ABB RAPID module: Rapid logo Inclinado.mod

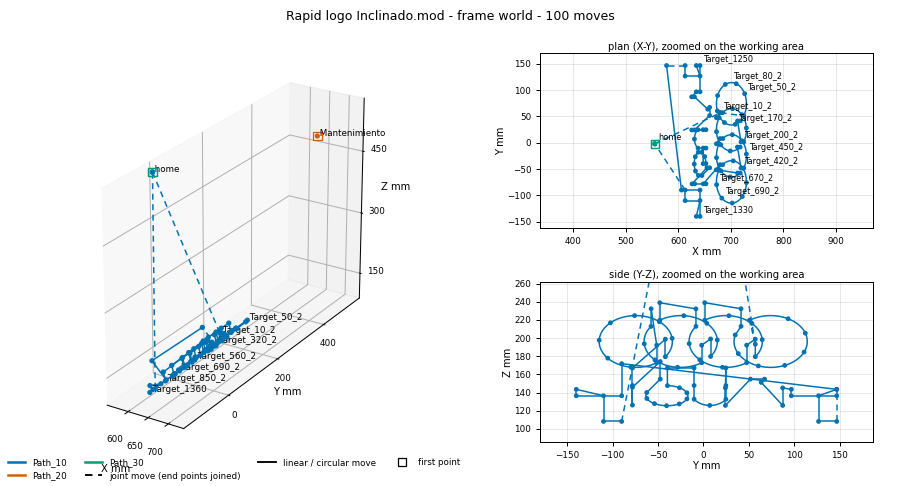
[picture p0: tool path of Rapid logo Inclinado.mod in frame world, 100 of 100 moves have a stored position in this frame; points joined in program order, loops and branches not executed]
MODULE Module1
    CONST robtarget Target_10_2:=[[-56.37355629,21.833194655,-12.40407904],[0.707106781,0,0,0.707106781],[0,0,-1,1],[9E+09,9E+09,9E+09,9E+09,9E+09,9E+09]];
    CONST robtarget Target_20_2:=[[-50.227,-27.838086869,0.000707115],[0.707106781,0,0,0.707106781],[0,0,-1,1],[9E+09,9E+09,9E+09,9E+09,9E+09,9E+09]];
    CONST robtarget Target_30_2:=[[-50.227,-27.838316171,0.001135326],[0.707106781,0,0,0.707106781],[0,0,-1,1],[9E+09,9E+09,9E+09,9E+09,9E+09,9E+09]];
    CONST robtarget Target_40_2:=[[-78.443,-34.755674334,0.002156228],[0.707106781,0,0,0.707106781],[0,0,-1,1],[9E+09,9E+09,9E+09,9E+09,9E+09,9E+09]];
    CONST robtarget Target_50_2:=[[-92.484,-30.22935476,0.001816803],[0.707106781,0,0,0.707106781],[0,0,-1,1],[9E+09,9E+09,9E+09,9E+09,9E+09,9E+09]];
    CONST robtarget Target_60_2:=[[-104.135,-20.748420193,0.00095273],[0.707106781,0,0,0.707106781],[0,0,-1,1],[9E+09,9E+09,9E+09,9E+09,9E+09,9E+09]];
    CONST robtarget Target_70_2:=[[-111.492,-7.712859409,0.000760167],[0.707106781,0,0,0.707106781],[0,0,-1,1],[9E+09,9E+09,9E+09,9E+09,9E+09,9E+09]];
    CONST robtarget Target_80_2:=[[-113.551,7.814084168,-0.000316037],[0.707106781,0,0,0.707106781],[0,0,-1,1],[9E+09,9E+09,9E+09,9E+09,9E+09,9E+09]];
    CONST robtarget Target_90_2:=[[-110.107,21.743448618,-0.000425835],[0.707106781,0,0,0.707106781],[0,0,-1,1],[9E+09,9E+09,9E+09,9E+09,9E+09,9E+09]];
    CONST robtarget Target_100_2:=[[-101.518,34.06976979,-0.001033142],[0.707106781,0,0,0.707106781],[0,0,-1,1],[9E+09,9E+09,9E+09,9E+09,9E+09,9E+09]];
    CONST robtarget Target_110_2:=[[-88.877,42.457578322,-0.001209673],[0.707106781,0,0,0.707106781],[0,0,-1,1],[9E+09,9E+09,9E+09,9E+09,9E+09,9E+09]];
    CONST robtarget Target_120_2:=[[-75.046,45.550294377,-0.000574222],[0.707106781,0,0,0.707106781],[0,0,-1,1],[9E+09,9E+09,9E+09,9E+09,9E+09,9E+09]];
    CONST robtarget Target_130_2:=[[-59.737,43.24160957,-0.001254548],[0.707106781,0,0,0.707106781],[0,0,-1,1],[9E+09,9E+09,9E+09,9E+09,9E+09,9E+09]];
    CONST robtarget Target_140_2:=[[-46.87,35.727016258,-0.000654802],[0.707106781,0,0,0.707106781],[0,0,-1,1],[9E+09,9E+09,9E+09,9E+09,9E+09,9E+09]];
    CONST robtarget Target_150_2:=[[-37.62,24.074953917,-0.00022001],[0.707106781,0,0,0.707106781],[0,0,-1,1],[9E+09,9E+09,9E+09,9E+09,9E+09,9E+09]];
    CONST robtarget Target_160_2:=[[-33.231,9.934106808,-0.000401667],[0.707106781,0,0,0.707106781],[0,0,-1,1],[9E+09,9E+09,9E+09,9E+09,9E+09,9E+09]];
    CONST robtarget Target_170_2:=[[-34.268,-4.941898461,0.000110514],[0.707106781,0,0,0.707106781],[0,0,-1,1],[9E+09,9E+09,9E+09,9E+09,9E+09,9E+09]];
    CONST robtarget Target_180_2:=[[-40.693,-18.501236857,0.089106304],[0.707106781,0,0,0.707106781],[0,0,-1,1],[9E+09,9E+09,9E+09,9E+09,9E+09,9E+09]];
    CONST robtarget Target_190_2:=[[-40.659,-28.454720515,-17.319460468],[0.707106781,0,0,0.707106781],[0,0,-1,1],[9E+09,9E+09,9E+09,9E+09,9E+09,9E+09]];
    CONST robtarget Target_200_2:=[[-0.697,-37.838908963,-17.319030487],[0.707106781,0,0,0.707106781],[0,0,-1,1],[9E+09,9E+09,9E+09,9E+09,9E+09,9E+09]];
    CONST robtarget Target_210_2:=[[-0.697,-27.838316171,0.001135326],[0.707106781,0,0,0.707106781],[0,0,-1,1],[9E+09,9E+09,9E+09,9E+09,9E+09,9E+09]];
    CONST robtarget Target_220_2:=[[-13.615,-33.787079032,0.001779373],[0.707106781,0,0,0.707106781],[0,0,-1,1],[9E+09,9E+09,9E+09,9E+09,9E+09,9E+09]];
    CONST robtarget Target_230_2:=[[-27.286,-34.931310202,0.001952004],[0.707106781,0,0,0.707106781],[0,0,-1,1],[9E+09,9E+09,9E+09,9E+09,9E+09,9E+09]];
    CONST robtarget Target_240_2:=[[-41.038,-31.199816129,0.000961671],[0.707106781,0,0,0.707106781],[0,0,-1,1],[9E+09,9E+09,9E+09,9E+09,9E+09,9E+09]];
    CONST robtarget Target_250_2:=[[-52.601,-22.954894729,0.001302226],[0.707106781,0,0,0.707106781],[0,0,-1,1],[9E+09,9E+09,9E+09,9E+09,9E+09,9E+09]];
    CONST robtarget Target_260_2:=[[-60.575,-11.244165105,0.000480163],[0.707106781,0,0,0.707106781],[0,0,-1,1],[9E+09,9E+09,9E+09,9E+09,9E+09,9E+09]];
    CONST robtarget Target_270_2:=[[-63.996,2.327231469,0.000364069],[0.707106781,0,0,0.707106781],[0,0,-1,1],[9E+09,9E+09,9E+09,9E+09,9E+09,9E+09]];
    CONST robtarget Target_280_2:=[[-62.487,16.549566353,-0.000316047],[0.707106781,0,0,0.707106781],[0,0,-1,1],[9E+09,9E+09,9E+09,9E+09,9E+09,9E+09]];
    CONST robtarget Target_290_2:=[[-56.39,28.971767635,-0.000857416],[0.707106781,0,0,0.707106781],[0,0,-1,1],[9E+09,9E+09,9E+09,9E+09,9E+09,9E+09]];
    CONST robtarget Target_300_2:=[[-56.367,19.00342355,-17.321167927],[0.707106781,0,0,0.707106781],[0,0,-1,1],[9E+09,9E+09,9E+09,9E+09,9E+09,9E+09]];
    CONST robtarget Target_310_2:=[[-46.834,28.340604975,-17.321014884],[0.707106781,0,0,0.707106781],[0,0,-1,1],[9E+09,9E+09,9E+09,9E+09,9E+09,9E+09]];
    CONST robtarget Target_320_2:=[[-46.834,38.341197767,-0.00084907],[0.707106781,0,0,0.707106781],[0,0,-1,1],[9E+09,9E+09,9E+09,9E+09,9E+09,9E+09]];
    CONST robtarget Target_330_2:=[[-33.859,44.305218974,-0.001065436],[0.707106781,0,0,0.707106781],[0,0,-1,1],[9E+09,9E+09,9E+09,9E+09,9E+09,9E+09]];
    CONST robtarget Target_340_2:=[[-20.239,45.433325791,-0.001165718],[0.707106781,0,0,0.707106781],[0,0,-1,1],[9E+09,9E+09,9E+09,9E+09,9E+09,9E+09]];
    CONST robtarget Target_350_2:=[[-6.223,41.574568908,-0.000596655],[0.707106781,0,0,0.707106781],[0,0,-1,1],[9E+09,9E+09,9E+09,9E+09,9E+09,9E+09]];
    CONST robtarget Target_360_2:=[[4.844,33.686749376,-0.000430885],[0.707106781,0,0,0.707106781],[-1,-1,0,1],[9E+09,9E+09,9E+09,9E+09,9E+09,9E+09]];
    CONST robtarget Target_370_2:=[[12.797,22.289578631,-0.000519591],[0.707106781,0,0,0.707106781],[-1,-1,0,1],[9E+09,9E+09,9E+09,9E+09,9E+09,9E+09]];
    CONST robtarget Target_380_2:=[[16.431,8.6200699,-0.000335384],[0.707106781,0,0,0.707106781],[-1,-1,0,1],[9E+09,9E+09,9E+09,9E+09,9E+09,9E+09]];
    CONST robtarget Target_390_2:=[[14.958,-6.043086672,0.000834231],[0.707106781,0,0,0.707106781],[-1,-1,0,1],[9E+09,9E+09,9E+09,9E+09,9E+09,9E+09]];
    CONST robtarget Target_400_2:=[[8.986,-18.294616208,0.000981918],[0.707106781,0,0,0.707106781],[-1,-1,0,1],[9E+09,9E+09,9E+09,9E+09,9E+09,9E+09]];
    CONST robtarget Target_410_2:=[[9.008,-28.264326332,-17.319694571],[0.707106781,0,0,0.707106781],[-1,-1,0,1],[9E+09,9E+09,9E+09,9E+09,9E+09,9E+09]];
    CONST robtarget Target_420_2:=[[48.833,-37.838908963,-17.319030487],[0.707106781,0,0,0.707106781],[-1,-1,0,1],[9E+09,9E+09,9E+09,9E+09,9E+09,9E+09]];
    CONST robtarget Target_430_2:=[[48.833,-27.838316171,0.001135326],[0.707106781,0,0,0.707106781],[-1,-1,0,1],[9E+09,9E+09,9E+09,9E+09,9E+09,9E+09]];
    CONST robtarget Target_440_2:=[[36.191,-33.714519443,0.001453804],[0.707106781,0,0,0.707106781],[-1,-1,0,1],[9E+09,9E+09,9E+09,9E+09,9E+09,9E+09]];
    CONST robtarget Target_450_2:=[[22.379,-34.942970463,0.00175625],[0.707106781,0,0,0.707106781],[-1,-1,0,1],[9E+09,9E+09,9E+09,9E+09,9E+09,9E+09]];
    CONST robtarget Target_460_2:=[[8.645,-31.272375718,0.001287239],[0.707106781,0,0,0.707106781],[-1,-1,0,1],[9E+09,9E+09,9E+09,9E+09,9E+09,9E+09]];
    CONST robtarget Target_470_2:=[[-2.93,-23.098281891,0.000953305],[0.707106781,0,0,0.707106781],[0,0,-1,1],[9E+09,9E+09,9E+09,9E+09,9E+09,9E+09]];
    CONST robtarget Target_480_2:=[[-10.814,-11.750850244,0.000893078],[0.707106781,0,0,0.707106781],[0,0,-1,1],[9E+09,9E+09,9E+09,9E+09,9E+09,9E+09]];
    CONST robtarget Target_490_2:=[[-14.498,2.811096116,0.000425657],[0.707106781,0,0,0.707106781],[0,0,-1,1],[9E+09,9E+09,9E+09,9E+09,9E+09,9E+09]];
    CONST robtarget Target_500_2:=[[-13.011,16.365002299,0.000015933],[0.707106781,0,0,0.707106781],[0,0,-1,1],[9E+09,9E+09,9E+09,9E+09,9E+09,9E+09]];
    CONST robtarget Target_510_2:=[[-7.137,28.586515175,-0.000121108],[0.707106781,0,0,0.707106781],[0,0,-1,1],[9E+09,9E+09,9E+09,9E+09,9E+09,9E+09]];
    CONST robtarget Target_520_2:=[[-7.137,18.585922383,-17.320286922],[0.707106781,0,0,0.707106781],[0,0,-1,1],[9E+09,9E+09,9E+09,9E+09,9E+09,9E+09]];
    CONST robtarget Target_530_2:=[[2.696,28.340604975,-17.321014884],[0.707106781,0,0,0.707106781],[0,0,-1,1],[9E+09,9E+09,9E+09,9E+09,9E+09,9E+09]];
    CONST robtarget Target_540_2:=[[2.696,38.341197767,-0.00084907],[0.707106781,0,0,0.707106781],[0,0,-1,1],[9E+09,9E+09,9E+09,9E+09,9E+09,9E+09]];
    CONST robtarget Target_550_2:=[[14.997,44.124253005,-0.000501529],[0.707106781,0,0,0.707106781],[-1,-1,0,1],[9E+09,9E+09,9E+09,9E+09,9E+09,9E+09]];
    CONST robtarget Target_560_2:=[[29.288,45.434191799,-0.001665747],[0.707106781,0,0,0.707106781],[-1,-1,0,1],[9E+09,9E+09,9E+09,9E+09,9E+09,9E+09]];
    CONST robtarget Target_570_2:=[[43.337,41.559310564,-0.001024336],[0.707106781,0,0,0.707106781],[-1,-1,0,1],[9E+09,9E+09,9E+09,9E+09,9E+09,9E+09]];
    CONST robtarget Target_580_2:=[[54.189,33.872679468,-0.000396886],[0.707106781,0,0,0.707106781],[-1,-1,0,1],[9E+09,9E+09,9E+09,9E+09,9E+09,9E+09]];
    CONST robtarget Target_590_2:=[[62.528,21.849622952,-0.000530122],[0.707106781,0,0,0.707106781],[-1,-1,0,1],[9E+09,9E+09,9E+09,9E+09,9E+09,9E+09]];
    CONST robtarget Target_600_2:=[[65.937,8.892951917,0.000300757],[0.707106781,0,0,0.707106781],[-1,-1,0,1],[9E+09,9E+09,9E+09,9E+09,9E+09,9E+09]];
    CONST robtarget Target_610_2:=[[64.517,-5.942742468,0.000632066],[0.707106781,0,0,0.707106781],[-1,-1,0,1],[9E+09,9E+09,9E+09,9E+09,9E+09,9E+09]];
    CONST robtarget Target_620_2:=[[58.496,-18.322400822,0.000858513],[0.707106781,0,0,0.707106781],[-1,-1,0,1],[9E+09,9E+09,9E+09,9E+09,9E+09,9E+09]];
    CONST robtarget Target_630_2:=[[58.383,-28.479773053,-17.318851916],[0.707106781,0,0,0.707106781],[-1,-1,0,1],[9E+09,9E+09,9E+09,9E+09,9E+09,9E+09]];
    CONST robtarget Target_640_2:=[[52.226,28.340604975,-17.321014884],[0.707106781,0,0,0.707106781],[-1,-1,0,1],[9E+09,9E+09,9E+09,9E+09,9E+09,9E+09]];
    CONST robtarget Target_650_2:=[[52.226,38.341197767,-0.00084907],[0.707106781,0,0,0.707106781],[-1,-1,0,1],[9E+09,9E+09,9E+09,9E+09,9E+09,9E+09]];
    CONST robtarget Target_660_2:=[[65.447,44.367484341,-0.001220779],[0.707106781,0,0,0.707106781],[-1,-1,0,1],[9E+09,9E+09,9E+09,9E+09,9E+09,9E+09]];
    CONST robtarget Target_670_2:=[[80.648,45.231271346,-0.001127368],[0.707106781,0,0,0.707106781],[-1,-1,0,1],[9E+09,9E+09,9E+09,9E+09,9E+09,9E+09]];
    CONST robtarget Target_680_2:=[[94.887,40.510959505,-0.000785768],[0.707106781,0,0,0.707106781],[-1,-1,0,1],[9E+09,9E+09,9E+09,9E+09,9E+09,9E+09]];
    CONST robtarget Target_690_2:=[[106.195,31.179608209,-0.000840934],[0.707106781,0,0,0.707106781],[-1,-1,0,1],[9E+09,9E+09,9E+09,9E+09,9E+09,9E+09]];
    CONST robtarget Target_700_2:=[[113.612,17.854675076,0.000153874],[0.707106781,0,0,0.707106781],[-1,-1,0,1],[9E+09,9E+09,9E+09,9E+09,9E+09,9E+09]];
    CONST robtarget Target_710_2:=[[115.581,3.23046335,0.000776639],[0.707106781,0,0,0.707106781],[-1,-1,0,1],[9E+09,9E+09,9E+09,9E+09,9E+09,9E+09]];
    CONST robtarget Target_720_2:=[[112.232,-10.957390781,0.001178007],[0.707106781,0,0,0.707106781],[-1,-1,0,1],[9E+09,9E+09,9E+09,9E+09,9E+09,9E+09]];
    CONST robtarget Target_730_2:=[[103.201,-23.874250963,0.000962006],[0.707106781,0,0,0.707106781],[-1,-1,0,1],[9E+09,9E+09,9E+09,9E+09,9E+09,9E+09]];
    CONST robtarget Target_740_2:=[[90.94,-31.928278149,0.001253355],[0.707106781,0,0,0.707106781],[-1,-1,0,1],[9E+09,9E+09,9E+09,9E+09,9E+09,9E+09]];
    CONST robtarget Target_750_2:=[[76.607,-35.064403142,0.001432857],[0.707106781,0,0,0.707106781],[-1,-1,0,1],[9E+09,9E+09,9E+09,9E+09,9E+09,9E+09]];
    CONST robtarget Target_760_2:=[[62.223,-32.908533711,0.001434457],[0.707106781,0,0,0.707106781],[-1,-1,0,1],[9E+09,9E+09,9E+09,9E+09,9E+09,9E+09]];
    CONST robtarget Target_770_2:=[[49.279,-25.574906369,0.001398618],[0.707106781,0,0,0.707106781],[-1,-1,0,1],[9E+09,9E+09,9E+09,9E+09,9E+09,9E+09]];
    CONST robtarget Target_780_2:=[[39.611,-13.556813975,0.000933947],[0.707106781,0,0,0.707106781],[-1,-1,0,1],[9E+09,9E+09,9E+09,9E+09,9E+09,9E+09]];
    CONST robtarget Target_790_2:=[[35.255,0.363122261,0.000494345],[0.707106781,0,0,0.707106781],[-1,-1,0,1],[9E+09,9E+09,9E+09,9E+09,9E+09,9E+09]];
    CONST robtarget Target_800_2:=[[36.202,15.191620477,-0.00030082],[0.707106781,0,0,0.707106781],[-1,-1,0,1],[9E+09,9E+09,9E+09,9E+09,9E+09,9E+09]];
    CONST robtarget Target_810_2:=[[42.65,28.945349059,-0.000614842],[0.707106781,0,0,0.707106781],[-1,-1,0,1],[9E+09,9E+09,9E+09,9E+09,9E+09,9E+09]];
    CONST robtarget Target_820_2:=[[42.65,18.944756267,-17.320780656],[0.707106781,0,0,0.707106781],[-1,-1,0,1],[9E+09,9E+09,9E+09,9E+09,9E+09,9E+09]];
    CONST robtarget Target_830_2:=[[78.968,63.836225874,-17.322010862],[0.707106781,0,0,0.707106781],[-1,-1,0,1],[9E+09,9E+09,9E+09,9E+09,9E+09,9E+09]];
    CONST robtarget Target_840_2:=[[78.968,73.836818666,-0.001845049],[0.707106781,0,0,0.707106781],[-1,-1,0,1],[9E+09,9E+09,9E+09,9E+09,9E+09,9E+09]];
    CONST robtarget Target_850_2:=[[78.968,104.377324543,-0.003182388],[0.707106781,0,0,0.707106781],[-1,-1,0,1],[9E+09,9E+09,9E+09,9E+09,9E+09,9E+09]];
    CONST robtarget Target_860_2:=[[78.968,93.82340557,-17.323718301],[0.707106781,0,0,0.707106781],[-1,-1,0,1],[9E+09,9E+09,9E+09,9E+09,9E+09,9E+09]];
    CONST robtarget Target_870_2:=[[48.351,53.873158678,-17.322208436],[0.707106781,0,0,0.707106781],[-1,-1,0,1],[9E+09,9E+09,9E+09,9E+09,9E+09,9E+09]];
    CONST robtarget Target_880_2:=[[48.351,63.87375147,-0.002042622],[0.707106781,0,0,0.707106781],[-1,-1,0,1],[9E+09,9E+09,9E+09,9E+09,9E+09,9E+09]];
    CONST robtarget Target_890_2:=[[63.169,84.713777945,-0.002771169],[0.707106781,0,0,0.707106781],[-1,-1,0,1],[9E+09,9E+09,9E+09,9E+09,9E+09,9E+09]];
    CONST robtarget Target_900_2:=[[64.162,89.365128281,-0.002555273],[0.707106781,0,0,0.707106781],[-1,-1,0,1],[9E+09,9E+09,9E+09,9E+09,9E+09,9E+09]];
    CONST robtarget Target_910_2:=[[63.046,94.05095937,-0.002618126],[0.707106781,0,0,0.707106781],[-1,-1,0,1],[9E+09,9E+09,9E+09,9E+09,9E+09,9E+09]];
    CONST robtarget Target_920_2:=[[59.797,98.451382173,-0.003012843],[0.707106781,0,0,0.707106781],[-1,-1,0,1],[9E+09,9E+09,9E+09,9E+09,9E+09,9E+09]];
    CONST robtarget Target_930_2:=[[54.654,102.034659013,-0.002717958],[0.707106781,0,0,0.707106781],[-1,-1,0,1],[9E+09,9E+09,9E+09,9E+09,9E+09,9E+09]];
    CONST robtarget Target_940_2:=[[48.275,104.357602106,-0.003341967],[0.707106781,0,0,0.707106781],[-1,-1,0,1],[9E+09,9E+09,9E+09,9E+09,9E+09,9E+09]];
    CONST robtarget Target_950_2:=[[41.357,105.262200024,-0.002563419],[0.707106781,0,0,0.707106781],[-1,-1,0,1],[9E+09,9E+09,9E+09,9E+09,9E+09,9E+09]];
    CONST robtarget Target_960_2:=[[33.909,104.634948216,-0.002973928],[0.707106781,0,0,0.707106781],[-1,-1,0,1],[9E+09,9E+09,9E+09,9E+09,9E+09,9E+09]];
    CONST robtarget Target_970_2:=[[27.402,102.507729408,-0.003352153],[0.707106781,0,0,0.707106781],[-1,-1,0,1],[9E+09,9E+09,9E+09,9E+09,9E+09,9E+09]];
    CONST robtarget Target_980_2:=[[22.063,98.927184643,-0.002915081],[0.707106781,0,0,0.707106781],[-1,-1,0,1],[9E+09,9E+09,9E+09,9E+09,9E+09,9E+09]];
    CONST robtarget Target_990_2:=[[18.943,94.70772781,-0.003084271],[0.707106781,0,0,0.707106781],[-1,-1,0,1],[9E+09,9E+09,9E+09,9E+09,9E+09,9E+09]];
    CONST robtarget Target_1000_2:=[[17.87,89.969059568,-0.002536271],[0.707106781,0,0,0.707106781],[-1,-1,0,1],[9E+09,9E+09,9E+09,9E+09,9E+09,9E+09]];
    CONST robtarget Target_1010_2:=[[18.988,85.194544537,-0.002075501],[0.707106781,0,0,0.707106781],[-1,-1,0,1],[9E+09,9E+09,9E+09,9E+09,9E+09,9E+09]];
    CONST robtarget Target_1020_2:=[[22.223,80.811112095,-0.002253162],[0.707106781,0,0,0.707106781],[-1,-1,0,1],[9E+09,9E+09,9E+09,9E+09,9E+09,9E+09]];
    CONST robtarget Target_1030_2:=[[27.118,77.349267934,-0.002224654],[0.707106781,0,0,0.707106781],[-1,-1,0,1],[9E+09,9E+09,9E+09,9E+09,9E+09,9E+09]];
    CONST robtarget Target_1040_2:=[[33.511,74.951899184,-0.002507063],[0.707106781,0,0,0.707106781],[-1,-1,0,1],[9E+09,9E+09,9E+09,9E+09,9E+09,9E+09]];
    CONST robtarget Target_1050_2:=[[40.419,73.994964144,-0.001934454],[0.707106781,0,0,0.707106781],[-1,-1,0,1],[9E+09,9E+09,9E+09,9E+09,9E+09,9E+09]];
    CONST robtarget Target_1060_2:=[[40.491,63.992139305,-17.321966217],[0.707106781,0,0,0.707106781],[-1,-1,0,1],[9E+09,9E+09,9E+09,9E+09,9E+09,9E+09]];
    CONST robtarget Target_1070_2:=[[11.022,63.836225874,-17.322010862],[0.707106781,0,0,0.707106781],[-1,-1,0,1],[9E+09,9E+09,9E+09,9E+09,9E+09,9E+09]];
    CONST robtarget Target_1080_2:=[[11.022,73.836818666,-0.001845049],[0.707106781,0,0,0.707106781],[-1,-1,0,1],[9E+09,9E+09,9E+09,9E+09,9E+09,9E+09]];
    CONST robtarget Target_1090_2:=[[11.022,95.187128364,-0.002754582],[0.707106781,0,0,0.707106781],[-1,-1,0,1],[9E+09,9E+09,9E+09,9E+09,9E+09,9E+09]];
    CONST robtarget Target_1100_2:=[[3.873,102.062443627,-0.002594553],[0.707106781,0,0,0.707106781],[-1,-1,0,1],[9E+09,9E+09,9E+09,9E+09,9E+09,9E+09]];
    CONST robtarget Target_1110_2:=[[-6.178,104.834770614,-0.002878227],[0.707106781,0,0,0.707106781],[0,0,-1,1],[9E+09,9E+09,9E+09,9E+09,9E+09,9E+09]];
    CONST robtarget Target_1120_2:=[[-16.254,102.380966628,-0.002907415],[0.707106781,0,0,0.707106781],[0,0,-1,1],[9E+09,9E+09,9E+09,9E+09,9E+09,9E+09]];
    CONST robtarget Target_1130_2:=[[-23.975,95.187128364,-0.002754582],[0.707106781,0,0,0.707106781],[0,0,-1,1],[9E+09,9E+09,9E+09,9E+09,9E+09,9E+09]];
    CONST robtarget Target_1140_2:=[[-23.975,73.836818666,-0.001845049],[0.707106781,0,0,0.707106781],[0,0,-1,1],[9E+09,9E+09,9E+09,9E+09,9E+09,9E+09]];
    CONST robtarget Target_1150_2:=[[-23.975,63.836225874,-17.322010862],[0.707106781,0,0,0.707106781],[0,0,-1,1],[9E+09,9E+09,9E+09,9E+09,9E+09,9E+09]];
    CONST robtarget Target_1160_2:=[[-23.471,94.836409868,-17.323178091],[0.707106781,0,0,0.707106781],[0,0,-1,1],[9E+09,9E+09,9E+09,9E+09,9E+09,9E+09]];
    CONST robtarget Target_1170_2:=[[-23.471,104.83700266,-0.003012278],[0.707106781,0,0,0.707106781],[0,0,-1,1],[9E+09,9E+09,9E+09,9E+09,9E+09,9E+09]];
    CONST robtarget Target_1180_2:=[[-51.009,63.87375147,-0.002042622],[0.707106781,0,0,0.707106781],[0,0,-1,1],[9E+09,9E+09,9E+09,9E+09,9E+09,9E+09]];
    CONST robtarget Target_1190_2:=[[-66.555,63.87375147,-0.002042622],[0.707106781,0,0,0.707106781],[0,0,-1,1],[9E+09,9E+09,9E+09,9E+09,9E+09,9E+09]];
    CONST robtarget Target_1200_2:=[[-62.898,68.923380565,-0.002001302],[0.707106781,0,0,0.707106781],[0,0,-1,1],[9E+09,9E+09,9E+09,9E+09,9E+09,9E+09]];
    CONST robtarget Target_1210_2:=[[-86.555,104.83700266,-0.003012278],[0.707106781,0,0,0.707106781],[0,0,-1,1],[9E+09,9E+09,9E+09,9E+09,9E+09,9E+09]];
    CONST robtarget Target_1220_2:=[[-86.555,94.836409868,-17.323178091],[0.707106781,0,0,0.707106781],[0,0,-1,1],[9E+09,9E+09,9E+09,9E+09,9E+09,9E+09]];
    CONST robtarget Target_1230:=[[-96.081,89.782,-10],[0.707106781,0,0,0.707106781],[0,0,-1,1],[9E+09,9E+09,9E+09,9E+09,9E+09,9E+09]];
    CONST robtarget Target_1240:=[[-96.081,89.782,0],[0.707106781,0,0,0.707106781],[0,0,-1,1],[9E+09,9E+09,9E+09,9E+09,9E+09,9E+09]];
    CONST robtarget Target_1250:=[[-146.081,89.782,0],[0.707106781,0,0,0.707106781],[0,0,-1,1],[9E+09,9E+09,9E+09,9E+09,9E+09,9E+09]];
    CONST robtarget Target_1260:=[[-146.081,89.782,-10],[0.707106781,0,0,0.707106781],[0,0,-1,1],[9E+09,9E+09,9E+09,9E+09,9E+09,9E+09]];
    CONST robtarget Target_1270:=[[-126.081,89.782,0],[0.707106781,0,0,0.707106781],[0,0,-1,1],[9E+09,9E+09,9E+09,9E+09,9E+09,9E+09]];
    CONST robtarget Target_1280:=[[-126.081,129.782,0],[0.707106781,0,0,0.707106781],[0,0,-1,1],[9E+09,9E+09,9E+09,9E+09,9E+09,9E+09]];
    CONST robtarget Target_1290:=[[-146.081,129.782,0],[0.707106781,0,0,0.707106781],[0,0,-1,1],[9E+09,9E+09,9E+09,9E+09,9E+09,9E+09]];
    CONST robtarget Target_1300:=[[-146.081,129.782,-50],[0.707106781,0,0,0.707106781],[0,0,-1,1],[9E+09,9E+09,9E+09,9E+09,9E+09,9E+09]];
    CONST robtarget Target_1310:=[[90.838,89.782,-50],[0.707106781,0,0,0.707106781],[-1,-1,0,1],[9E+09,9E+09,9E+09,9E+09,9E+09,9E+09]];
    CONST robtarget Target_1320:=[[90.838,89.782,0],[0.707106781,0,0,0.707106781],[-1,-1,0,1],[9E+09,9E+09,9E+09,9E+09,9E+09,9E+09]];
    CONST robtarget Target_1330:=[[140.838,89.782,0],[0.707106781,0,0,0.707106781],[-1,-1,0,1],[9E+09,9E+09,9E+09,9E+09,9E+09,9E+09]];
    CONST robtarget Target_1340:=[[140.838,89.782,-10],[0.707106781,0,0,0.707106781],[-1,-1,0,1],[9E+09,9E+09,9E+09,9E+09,9E+09,9E+09]];
    CONST robtarget Target_1350:=[[110.838,89.782,0],[0.707106781,0,0,0.707106781],[-1,-1,0,1],[9E+09,9E+09,9E+09,9E+09,9E+09,9E+09]];
    CONST robtarget Target_1360:=[[110.838,129.782,0],[0.707106781,0,0,0.707106781],[-1,-1,0,1],[9E+09,9E+09,9E+09,9E+09,9E+09,9E+09]];
    CONST robtarget Target_1370:=[[90.838,129.782,0],[0.707106781,0,0,0.707106781],[-1,-1,0,1],[9E+09,9E+09,9E+09,9E+09,9E+09,9E+09]];
    CONST robtarget home:=[[2.874,-145.21377629,-356.72517815],[0.683012702,-0.183012701,0.183012701,0.683012702],[-1,0,-1,0],[9E+09,9E+09,9E+09,9E+09,9E+09,9E+09]];
    CONST robtarget Mantenimiento:=[[-531.736245023,-148.098354507,-242.688419489],[0.851265704,-0.292898067,0.051053304,0.432378287],[0,0,-1,0],[9E+09,9E+09,9E+09,9E+09,9E+09,9E+09]];
    PERS tooldata Herramienta1:=[TRUE,[[83.437,-2.036,104.634],[0.923879533,0,0.382683432,0]],[0.3,[0,0,1],[1,0,0,0],0,0,0]];
    TASK PERS wobjdata AUDI:=[FALSE,TRUE,"",[[704.75,0.838,150],[0.27059805,-0.653281482,0.653281482,-0.27059805]],[[0,-35.355339069,-35.355339049],[1,0,0,0]]];
    PROC Path_10()
        MoveL home,v100,z0,Herramienta1\WObj:=AUDI;
        MoveJ Target_10_2,v100,z5,Herramienta1\WObj:=AUDI;
        MoveJ Target_20_2,v100,fine,Herramienta1\WObj:=AUDI;
        MoveJ Target_30_2,v100,fine,Herramienta1\WObj:=AUDI;
        MoveC Target_40_2,Target_50_2,v100,z0,Herramienta1\WObj:=AUDI;
        MoveC Target_60_2,Target_70_2,v100,z0,Herramienta1\WObj:=AUDI;
        MoveC Target_80_2,Target_90_2,v100,z0,Herramienta1\WObj:=AUDI;
        MoveC Target_100_2,Target_110_2,v100,z0,Herramienta1\WObj:=AUDI;
        MoveC Target_120_2,Target_130_2,v100,z0,Herramienta1\WObj:=AUDI;
        MoveC Target_140_2,Target_150_2,v100,z0,Herramienta1\WObj:=AUDI;
        MoveC Target_160_2,Target_170_2,v100,z0,Herramienta1\WObj:=AUDI;
        MoveL Target_180_2,v100,z0,Herramienta1\WObj:=AUDI;
        MoveL Target_190_2,v100,z0,Herramienta1\WObj:=AUDI;
        MoveL Target_200_2,v100,z0,Herramienta1\WObj:=AUDI;
        MoveL Target_210_2,v100,z0,Herramienta1\WObj:=AUDI;
        MoveC Target_220_2,Target_230_2,v100,z0,Herramienta1\WObj:=AUDI;
        MoveC Target_240_2,Target_250_2,v100,z0,Herramienta1\WObj:=AUDI;
        MoveC Target_260_2,Target_270_2,v100,z0,Herramienta1\WObj:=AUDI;
        MoveC Target_280_2,Target_290_2,v100,z0,Herramienta1\WObj:=AUDI;
        MoveL Target_300_2,v100,z0,Herramienta1\WObj:=AUDI;
        MoveL Target_310_2,v100,z0,Herramienta1\WObj:=AUDI;
        MoveL Target_320_2,v100,z0,Herramienta1\WObj:=AUDI;
        MoveC Target_330_2,Target_340_2,v100,z0,Herramienta1\WObj:=AUDI;
        MoveC Target_350_2,Target_360_2,v100,z0,Herramienta1\WObj:=AUDI;
        MoveC Target_370_2,Target_380_2,v100,z0,Herramienta1\WObj:=AUDI;
        MoveC Target_390_2,Target_400_2,v100,z0,Herramienta1\WObj:=AUDI;
        MoveL Target_410_2,v100,z0,Herramienta1\WObj:=AUDI;
        MoveL Target_420_2,v100,z0,Herramienta1\WObj:=AUDI;
        MoveL Target_430_2,v100,z0,Herramienta1\WObj:=AUDI;
        MoveC Target_440_2,Target_450_2,v100,z0,Herramienta1\WObj:=AUDI;
        MoveC Target_460_2,Target_470_2,v100,z0,Herramienta1\WObj:=AUDI;
        MoveC Target_480_2,Target_490_2,v100,z0,Herramienta1\WObj:=AUDI;
        MoveC Target_500_2,Target_510_2,v100,z0,Herramienta1\WObj:=AUDI;
        MoveL Target_520_2,v100,z0,Herramienta1\WObj:=AUDI;
        MoveL Target_530_2,v100,z0,Herramienta1\WObj:=AUDI;
        MoveL Target_540_2,v100,z0,Herramienta1\WObj:=AUDI;
        MoveC Target_550_2,Target_560_2,v100,z0,Herramienta1\WObj:=AUDI;
        MoveC Target_570_2,Target_580_2,v100,z0,Herramienta1\WObj:=AUDI;
        MoveC Target_590_2,Target_600_2,v100,z0,Herramienta1\WObj:=AUDI;
        MoveC Target_610_2,Target_620_2,v100,z0,Herramienta1\WObj:=AUDI;
        MoveL Target_630_2,v100,z0,Herramienta1\WObj:=AUDI;
        MoveL Target_640_2,v100,z0,Herramienta1\WObj:=AUDI;
        MoveL Target_650_2,v100,z0,Herramienta1\WObj:=AUDI;
        MoveC Target_660_2,Target_670_2,v100,z0,Herramienta1\WObj:=AUDI;
        MoveC Target_680_2,Target_690_2,v100,z0,Herramienta1\WObj:=AUDI;
        MoveC Target_700_2,Target_710_2,v100,z0,Herramienta1\WObj:=AUDI;
        MoveC Target_720_2,Target_730_2,v100,z0,Herramienta1\WObj:=AUDI;
        MoveC Target_740_2,Target_750_2,v100,z0,Herramienta1\WObj:=AUDI;
        MoveC Target_760_2,Target_770_2,v100,z0,Herramienta1\WObj:=AUDI;
        MoveC Target_780_2,Target_790_2,v100,z0,Herramienta1\WObj:=AUDI;
        MoveC Target_800_2,Target_810_2,v100,z0,Herramienta1\WObj:=AUDI;
        MoveL Target_820_2,v100,z0,Herramienta1\WObj:=AUDI;
        MoveL Target_830_2,v100,z0,Herramienta1\WObj:=AUDI;
        MoveL Target_840_2,v100,z0,Herramienta1\WObj:=AUDI;
        MoveL Target_850_2,v100,z0,Herramienta1\WObj:=AUDI;
        MoveL Target_860_2,v100,z0,Herramienta1\WObj:=AUDI;
        MoveL Target_870_2,v100,z0,Herramienta1\WObj:=AUDI;
        MoveL Target_880_2,v100,z0,Herramienta1\WObj:=AUDI;
        MoveL Target_890_2,v100,z0,Herramienta1\WObj:=AUDI;
        MoveC Target_900_2,Target_910_2,v100,z0,Herramienta1\WObj:=AUDI;
        MoveC Target_920_2,Target_930_2,v100,z0,Herramienta1\WObj:=AUDI;
        MoveC Target_940_2,Target_950_2,v100,z0,Herramienta1\WObj:=AUDI;
        MoveC Target_960_2,Target_970_2,v100,z0,Herramienta1\WObj:=AUDI;
        MoveC Target_980_2,Target_990_2,v100,z0,Herramienta1\WObj:=AUDI;
        MoveC Target_1000_2,Target_1010_2,v100,z0,Herramienta1\WObj:=AUDI;
        MoveC Target_1020_2,Target_1030_2,v100,z0,Herramienta1\WObj:=AUDI;
        MoveC Target_1040_2,Target_1050_2,v100,z0,Herramienta1\WObj:=AUDI;
        MoveL Target_1060_2,v100,z0,Herramienta1\WObj:=AUDI;
        MoveL Target_1070_2,v100,z0,Herramienta1\WObj:=AUDI;
        MoveL Target_1080_2,v100,z0,Herramienta1\WObj:=AUDI;
        MoveL Target_1090_2,v100,z0,Herramienta1\WObj:=AUDI;
        MoveC Target_1100_2,Target_1110_2,v100,z0,Herramienta1\WObj:=AUDI;
        MoveC Target_1120_2,Target_1130_2,v100,z0,Herramienta1\WObj:=AUDI;
        MoveL Target_1140_2,v100,z0,Herramienta1\WObj:=AUDI;
        MoveL Target_1150_2,v100,z0,Herramienta1\WObj:=AUDI;
        MoveL Target_1160_2,v100,z0,Herramienta1\WObj:=AUDI;
        MoveL Target_1170_2,v100,z0,Herramienta1\WObj:=AUDI;
        MoveL Target_1180_2,v100,z0,Herramienta1\WObj:=AUDI;
        MoveL Target_1190_2,v100,z0,Herramienta1\WObj:=AUDI;
        MoveL Target_1200_2,v100,z0,Herramienta1\WObj:=AUDI;
        MoveL Target_1210_2,v100,z0,Herramienta1\WObj:=AUDI;
        MoveL Target_1220_2,v100,z0,Herramienta1\WObj:=AUDI;
        MoveL Target_1230,v100,z0,Herramienta1\WObj:=AUDI;
        MoveL Target_1240,v100,z0,Herramienta1\WObj:=AUDI;
        MoveL Target_1250,v100,z0,Herramienta1\WObj:=AUDI;
        MoveL Target_1260,v100,z0,Herramienta1\WObj:=AUDI;
        MoveL Target_1270,v100,z0,Herramienta1\WObj:=AUDI;
        MoveL Target_1280,v100,z0,Herramienta1\WObj:=AUDI;
        MoveL Target_1290,v100,z0,Herramienta1\WObj:=AUDI;
        MoveJ Target_1300,v100,z0,Herramienta1\WObj:=AUDI;
        MoveL Target_1310,v100,z0,Herramienta1\WObj:=AUDI;
        MoveL Target_1320,v100,z0,Herramienta1\WObj:=AUDI;
        MoveL Target_1330,v100,z0,Herramienta1\WObj:=AUDI;
        MoveL Target_1340,v100,z0,Herramienta1\WObj:=AUDI;
        MoveL Target_1350,v100,z0,Herramienta1\WObj:=AUDI;
        MoveL Target_1360,v100,z0,Herramienta1\WObj:=AUDI;
        MoveL Target_1370,v100,z0,Herramienta1\WObj:=AUDI;
        MoveJ home,v100,z0,Herramienta1\WObj:=AUDI;
    ENDPROC
    PROC main()
        WHILE TRUE
        DO
            WaitDI DI_01,1;
            SetDO DO_01,1;
            WaitDI DI_01,1;
            SetDO DO_02,0;
            WaitDI DI_01,1;
            Path_10;

            WaitDI DI_02,1;
            SetDO DO_02,1;
            WaitDI DI_02,1;
            SetDO DO_01,0;
            WaitDI DI_02,1;
            Path_20;

            WaitDI DI_03,1;
            Path_30;
        ENDWHILE
    ENDPROC
    PROC Path_20()
        MoveJ Mantenimiento,v100,z0,Herramienta1\WObj:=AUDI;
    ENDPROC
    PROC Path_30()
        MoveJ home,v100,z0,Herramienta1\WObj:=AUDI;
    ENDPROC
ENDMODULE
